FUNCTION_BLOCK FB_Position IMPLEMENTS IPosition
VAR_INPUT
	Sensor: BOOL;
END_VAR
VAR_OUTPUT
	Actor: BOOL;
END_VAR
VAR
END_VAR

// Release Signal
Locked := FALSE;

{warning 'Methodenimplementierung hinzufügen'}
METHOD Lock : BOOL
Locked := TRUE;
END_METHOD

PROPERTY Locked : BOOL
GET
VAR_INST
	_locked: BOOL;
END_VAR
END_GET
END_PROPERTY

METHOD MoveTo : BOOL
Actor := NOT Reached AND NOT Locked;
END_METHOD

PROPERTY Moving : BOOL
GET
Moving := Actor;
END_GET
END_PROPERTY

PROPERTY Reached : BOOL
GET
Reached := Sensor;
END_GET
END_PROPERTY

END_FUNCTION_BLOCK

(* stored: Version 1.1.0.1, ProductVersion 3.1.4024.11
   POU FB_Position: Id {8542c028-d930-47c9-a51d-a0824c396aea}, SpecialFunc None
   Method Lock: Id {fd575375-4470-454a-bff5-6842db67970d}
   Property Locked: Id {a407b0b7-e753-4ac5-8d7a-ded34fa01ef7}
   Get Get: Id {2a9c4fa8-787e-424b-a196-a514d3077775}
   Method MoveTo: Id {5fd46933-d567-466c-aaca-90b6bfa22e96}
   Property Moving: Id {31d22de0-bded-42c8-a401-0a383ec84842}
   Get Get: Id {1da6f644-cfff-41e5-b3a2-03ed63d93a37}
   Property Reached: Id {fb261eb4-b23e-4b37-aacf-36fbb85ee092}
   Get Get: Id {d79ba9f9-0e8b-446d-b9d7-93deec4f9ff9} *)
